// TIA Portal V20 export
DATA_BLOCK "Settings"   // DB6
{ DB_Accessible_From_OPC_UA := 'FALSE' }
// stored: DBAccessibleFromOPCUA false, DBAccessibleFromWebserver false, MemoryReserve 100
   VAR
      diagPlc : "LAF_typePlcDiag";   // HMI interface PLC diag
      checksum : "LAF_typeChecksum";   // HMI interface PLCChecksum
      diagMemCard : "LAF_typeMemCardDiag";   // HMI interface SMCDiag
      cycleTimes : "LSicar_typeGlobalRuntime";
      setLocalPlcTime : "LAF_typeSetPlcTime";
      ITConnection : Bool := FALSE;   // Provides a visual representation of the connection with the IT systems.
   END_VAR
BEGIN
   diagPlc.im1PlantDesignLocIdent := 'GM BCDC';
   diagPlc.im1PlantDesignation := 'GM BCDC';
END_DATA_BLOCK
